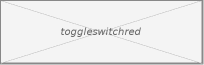
VISUALIZATION ToggleSwitch1  // 204x65
VAR_IN_OUT
	m_Input_Inst : None;
END_VAR
    Image (0,0 202x62), invisible if: (NOT m_Input_Inst) <> 0, image: toggleswitchgreen
        toggle m_Input_Inst
    Image (0,0 202x63), invisible if: (m_Input_Inst) <> 0, image: toggleswitchred
        toggle m_Input_Inst
END_VISUALIZATION

(* stored: Version 1.1.0.1, ProductVersion 3.1.4018.2
   Visu ToggleSwitch1: Id {7197957d-9b46-4213-9d7f-8c2ffb8ac790} *)
